# B&R Automation Studio project SDC_Encoder
Automation Studio 4.11.2.75; technology packages: Acp10Arnc0 5.22.1

## Configuration Config1

CPU X20CP1382, AutomationRuntime D4.26, Build 4.1.2, Safety 0.0, Vc V4.72.5

### Task classes (Cpu.sw)
```
Cyclic#1:
  ncsdcctrl <- ncsdcctrl.prg
NcDataObjects: acp10etxen <- acp10etxen.dob, gAxis01a <- gAxis01obj.gAxis01a.dob, gAxis01i <- gAxis01obj.gAxis01i.dob
Libraries: Acp10man, Acp10par, NcGlobal, Acp10sdc, Acp10_MC, sys_lib, brsystem, runtime, AsBrStr
```

### Hardware
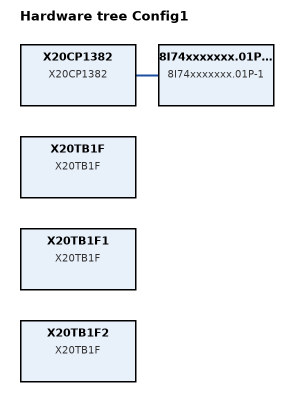
```
8I74xxxxxxx.01P-1 : 8I74xxxxxxx.01P-1 v1.6.2.0  [PLK1 -> X20CP1382.IF3 (NodeNumber=1) [Cable Type=PowerlinkCable, Length=10, Version=1.0.0.3]]
X20CP1382 : X20CP1382 v1.15.0.0  [X1 -> X1.SL; X2 -> X2.SL; X3 -> X3.SL]
  Module X1 (Type=X1, Virtual=true, Version=1.15.0.0)
    Connection (Connector=SS1, TargetModule=X20TB1F, TargetConnector=SS)
    Connection (Connector=SL, TargetModule=X20CP1382, TargetConnector=X1)
  Module X2 (Type=X2, Virtual=true, Version=1.15.0.0)
    Connection (Connector=SS1, TargetModule=X20TB1F1, TargetConnector=SS)
    Connection (Connector=SL, TargetModule=X20CP1382, TargetConnector=X2)
  Module X3 (Type=X3, Virtual=true, Version=1.15.0.0)
    Connection (Connector=SS1, TargetModule=X20TB1F2, TargetConnector=SS)
    Connection (Connector=SL, TargetModule=X20CP1382, TargetConnector=X3)
  Connector IF2:
    ActivateDevice = 1
  ConfigurationID = SDC_Encoder_Config1
  TimerDeviceType = EPLX2X
  TimerDevice = X20CP1382.IF3
  Cyclic1Tolerance = 0
  Cyclic1Output = 1
X20TB1F : X20TB1F v1.0.0.0
X20TB1F1 : X20TB1F v1.0.0.0
X20TB1F2 : X20TB1F v1.0.0.0
```

### IoMap.iom - X20CP1382/IoMap.iom
```iecst
VAR_CONFIG
	        Cyclic#1.gAxis01_DrvIf.iLifeCnt AT %IB."8I74xxxxxxx.01P-1".SDC_LifeCnt;
	        Cyclic#1.gAxis01_DrvIf.iDrvOK AT %IX."8I74xxxxxxx.01P-1".ETAD_Input_Bool_02;
	        Cyclic#1.gAxis01_DrvIf.oSetTime AT %QW."8I74xxxxxxx.01P-1".SDC_SetTime;
	        Cyclic#1.gAxis01_DrvIf.oSetPos AT %QW."8I74xxxxxxx.01P-1".LFRD_Output;
	        Cyclic#1.gAxis01_DiDoIf.iLifeCntDriveReady AT %IB."8I74xxxxxxx.01P-1".SDC_LifeCnt;
	        Cyclic#1.gAxis01_DiDoIf.iLifeCntDriveEnable AT %IB."8I74xxxxxxx.01P-1".SDC_LifeCnt;
	        Cyclic#1.gAxis01_DiDoIf.oDriveEnable AT %QX."8I74xxxxxxx.01P-1".CMDD_Output_Bool_00;
	        Cyclic#1.gAxis01_ModuleOk AT %QX."8I74xxxxxxx.01P-1".CMDD_Output_Bool_01;
	        Cyclic#1.gAxis01_ModuleOk AT %QX."8I74xxxxxxx.01P-1".CMDD_Output_Bool_02;
	        Cyclic#1.gAxis01_ModuleOk AT %IX."8I74xxxxxxx.01P-1".ModuleOk;
	        Cyclic#1.gAxis01_DiDoIf.oDriveEnable AT %QX."8I74xxxxxxx.01P-1".CMDD_Output_Bool_03;
	        Cyclic#1.gAxis01_DiDoIf.iDriveReady AT %IX."8I74xxxxxxx.01P-1".ETAD_Input_Bool_02;
END_VAR
```

### Acp10cfg.ncc - X20CP1382/Motion/Acp10cfg.ncc
```
NcConfiguration (Version=5.22.1, NcSwId=Acp10)
  ACP10CF1_typ:
    cnt_nettrc_rec_drive = 150
    bufsize_trace_upload = 1200
    tc_nc_man_task = Cyclic #1
    glob_pv_as_ncobject = Yes
    ncsys_dl_broadcast = Yes
    ncsys_dl_acp_reset = Yes
    safemc_log_err_to_ax = Yes
    network_init:
      ncsw_init_execute = Yes
      automatic_execute = No
      node_nr_warning = Yes
      net_err_before_ncact = Yes
    nettrc:
      enter_parsecrec = Yes
      enter_ncaction = Yes
      save_ring_startidx = No
    cam_prof_download:
      cam_dat_dl_parallel = No
      tc_cam_dl_parallel = Task class for NC Manager task
    sdc_if[0]:
      if_name = SDC_IF1
      mc_broadcast_size = 800
      mc_broadcast_extdat = No
```

### Acp10map.ncm - X20CP1382/Motion/Acp10map.ncm
```
NcMapping (NcSwId=Acp10)
  NcObject gAxis01 (ModuleId=8I74xxxxxxx.01P-1, ModuleAddress=SDC_IF1.ST1, Type=ncAXIS, Channel=1, AcoposSimulation=Off, InitParameter=gAxis01i, AcoposParameter=gAxis01a, Disabled=FALSE, ModuleDisabled=FALSE)
```

## Logical view

Binary libraries used (declarations not repeated): operator, runtime, astime, AsIecCon, Acp10man 5.22.1, Acp10par 5.22.1, NcGlobal 5.22.1, Acp10sdc 5.22.1, Acp10_MC 5.22.1, sys_lib, brsystem, AsBrStr

### Global.var - Global variables
```iecst
VAR
	gAxis01 : ACP10AXIS_typ;
	gAxis01_HW : SdcHwCfg_typ := (0);
	gAxis01_DrvIf : SdcDrvIf16_typ := (0);
	gAxis01_DiDoIf : SdcDiDoIf_typ := (0);
	gAxis01_ModuleOk : BOOL := 0;
	gAxis01_EncIF1 : SdcEncIf16_typ;
END_VAR
```


### Program Logical/ncsdcctrl (IEC)

#### ncsdcctrlCyclic.st
```iecst
PROGRAM _CYCLIC

(* ### BEGIN gAxis01 ### *)

(* life counter emulation of digital inputs *)
        gAxis01_DiDoIf.iLifeCntReference := gAxis01_DiDoIf.iLifeCntReference + 1;
        gAxis01_DiDoIf.iLifeCntNegHwEnd  := gAxis01_DiDoIf.iLifeCntNegHwEnd  + 1;
	gAxis01_DiDoIf.iLifeCntPosHwEnd  := gAxis01_DiDoIf.iLifeCntPosHwEnd  + 1;

	gAxis01_EncIF1.iLifeCnt := gAxis01_EncIF1.iLifeCnt +1;

//	ENCOD_OK := encoder's moduleOk
//	gAxis01_EncIF1.iActPos := Actual Position value
//	gAxis01_EncIF1.iActTime := ActTime;

(* ### END gAxis01 ### *)

END_PROGRAM
```

#### ncsdcctrlInit.st
```iecst
PROGRAM _INIT

(* ### BEGIN gAxis01 ### *)

(* initialize variables *)
        gAxis01_HW.DrvIf_Typ := ncSDC_DRVSERVO16;
        brsstrcpy(ADR(gAxis01_HW.DrvIf_Name[0]), ADR('gAxis01_DrvIf'));
        gAxis01_HW.DiDoIf_Typ := ncSDC_DIDO;
        brsstrcpy(ADR(gAxis01_HW.DiDoIf_Name[0]), ADR('gAxis01_DiDoIf'));

(* force variable offset generation *)
        gAxis01.size                      := gAxis01.size;
        gAxis01_DrvIf.iLifeCnt            := gAxis01_DrvIf.iLifeCnt;
        gAxis01_DiDoIf.iLifeCntDriveReady := gAxis01_DiDoIf.iLifeCntDriveReady;
		gAxis01_ModuleOk                  := gAxis01_ModuleOk;

	(*Encoder Addition*)
		gAxis01_EncIF1					:=	gAxis01_EncIF1;

(* assign your hardware inputs here*)

(*      gAxis01_DiDoIf.iPosHwEnd  := gAxis01_DiDoIf.iPosHwEnd;
        gAxis01_DiDoIf.iNegHwEnd  := gAxis01_DiDoIf.iNegHwEnd;
        gAxis01_DiDoIf.iReference := gAxis01_DiDoIf.iReference;
 *)

(* ### END gAxis01 ### *)

END_PROGRAM
```

#### ncsdcctrl.var
```iecst
VAR
	ENCOD_OK : BOOL;
END_VAR
```

### Data object Logical/acp10etxen (Ett)

- acp10etxen.ett (not shown)

### Package Logical/gAxis01obj - gAxis01obj

### gAxis01a.apt
```
AcoposParameterTable:
  Root Parameters:
    64201 = 546116.666666667 (Name=SERVO_V_MAX_OUTPUT)
```

### gAxis01i.ax
```
InitParameter (Version=5.22.1, NcSwId=Acp10)
  ACP10AXIS_typ:
    dig_in:
      level:
        reference = ncACTIV_HI
        pos_hw_end = ncACTIV_LO
        neg_hw_end = ncACTIV_LO
        trigger1 = ncACTIV_HI
        trigger2 = ncACTIV_LO + ncQUICKSTOP
    encoder_if:
      parameter:
        count_dir = ncSTANDARD
        scaling:
          load:
            units = 1000
            rev_motor = 1
    limit:
      parameter:
        v_pos = 10000
        v_neg = 10000
        a1_pos = 50000
        a2_pos = 50000
        a1_neg = 50000
        a2_neg = 50000
        t_jolt = 0
        t_in_pos = 0
        pos_sw_end = 2000000000
        neg_sw_end = -2000000000
        ds_warning = 500
        ds_stop = 1000
        a_stop = 1.0e30
        dv_stop = 0
        dv_stop_mode = ncOFF
    controller:
      mode = ncPOSITION
      position:
        kv = 50
        tn = 0
        t_predict = 0.05
        t_total = 0.05
        p_max = 1.0e30
        i_max = 0
      speed:
        kv = 2.0
        tn = 0
        t_filter = 0.0
        isq_filter1:
          type = ncOFF
          a0 = 0.0
          a1 = 0.0
          b0 = 0.0
          b1 = 0.0
          b2 = 0.0
          c0_par_id = 0
          c1_par_id = 0
        isq_filter2:
          type = ncOFF
          a0 = 0.0
          a1 = 0.0
          b0 = 0.0
          b1 = 0.0
          b2 = 0.0
          c0_par_id = 0
          c1_par_id = 0
        isq_filter3:
          type = ncOFF
          a0 = 0.0
          a1 = 0.0
          b0 = 0.0
          b1 = 0.0
          b2 = 0.0
          c0_par_id = 0
          c1_par_id = 0
      uf:
        type = ncLINEAR + ncCORRECTION
        auto_config = ncMOTOR_PAR
        u0 = 0
        un = 0
        fn = 50.0
        k_f_slip = 0
      ff:
        mode = ncSTANDARD
        torque_load = 0.0
        torque_pos = 0.0
        torque_neg = 0.0
        kv_torque = 0.0
        inertia = 0.0
        t_filter_a = 0.0
      fb:
        mode = ncSTANDARD
        speed_mix_ratio = 0.0
        speed_kv = 2.0
      model:
        mass1:
          inertia = 0
          viscous_friction = 0
        mass2:
          inertia = 0
          viscous_friction = 0
          stiffness = 0
          damping = 0
    move:
      stop:
        parameter[0]:
          decel_ramp = ncA_LIMIT
          controller = ncON
        parameter[1]:
          decel_ramp = ncA_LIMIT
          controller = ncON
        parameter[2]:
          decel_ramp = ncA_LIMIT
          controller = ncON
        parameter[3]:
          decel_ramp = ncA_LIMIT
          controller = ncON
        quickstop:
          decel_ramp = ncA_LIMIT
          t_jolt = 0
        drive_error:
          decel_ramp = ncA_LIMIT
      homing:
        parameter:
          s = 0
          v_switch = 5000
          v_trigger = 500
          a = 50000
          mode = ncDIRECT
          edge_sw = ncPOSITIVE
          start_dir = ncPOSITIVE
          trigg_dir = ncPOSITIVE
          ref_pulse = ncOFF
          fix_dir = ncOFF
          tr_s_block = 0
          torque_lim = 0
          ds_block = 0
          ds_stop = 0
      basis:
        parameter:
          v_pos = 5000
          v_neg = 5000
          a1_pos = 50000
          a2_pos = 50000
          a1_neg = 50000
          a2_neg = 50000
    message:
      text:
        parameter:
          format = ncBREAK
          columns = 80
          data_modul = acp10etxen
```

Listed in the project but not available here: Logical/Global.typ, Logical/ncsdcctrl/ncsdcctrl.typ
